// TwinCAT 3 PLC project Horiba
// Title: ZigaLibs.Horiba
// Company: Ziga Javornik
// Author: Ziga Javornik
// ProjectVersion: 0.0.1.0
// Description: Horiba EtherCAT device imeplementations library.
// ProgramVersion: 3.1.4024.0
// libraries:
//   Tc2_Standard, * (Beckhoff Automation GmbH)
//   Tc2_System, * (Beckhoff Automation GmbH)
//   Tc3_Module, * (Beckhoff Automation GmbH)
//   TcUnit, * (www.tcunit.org)
//   ZigaLibs.Automation, * (Ziga)
//   ZigaLibs.Core, * (Ziga)
//   ZigaLibs.Logging, * (Ziga)
// project tree:
//   SOURCE/MFC/SEC_ZXX7/DUTs/ E_SEC_ZXX7_ActuatorControl.TcDUT, E_SEC_ZXX7_ReadingStep.TcDUT, ST_SEC_ZXX7_ActiveExceptions.TcDUT, ST_SEC_ZXX7_CoeList.TcDUT, ST_SEC_ZXX7_Commands.TcDUT, ST_SEC_ZXX7_Feedback.TcDUT, ST_SEC_ZXX7_Inputs.TcDUT, ST_SEC_ZXX7_Outputs.TcDUT, T_SEC_ZXX7_ActiveExceptionStatus.TcDUT, T_SEC_ZXXX7_RampTime.TcDUT
//   SOURCE/MFC/SEC_ZXX7/POUs/ FB_MFC_SEC_ZXX7.TcPOU
//   TESTS/ PRG_TESTS.TcPOU
//   TESTS/Test suites/ FB_SUT_Tests.TcPOU (not stored)
// (motion and I/O tree: see PLC project logging)
// real-time tasks:
//   TASK TestsTask: cycle T#10ms, priority 20, ADS port 350
//   TASK PlcTask: cycle T#10ms, priority 21, ADS port 351

// ---- SOURCE/MFC/SEC_ZXX7/DUTs/E_SEC_ZXX7_ActuatorControl.TcDUT
{attribute 'qualified_only'}
{attribute 'strict'}
TYPE E_SEC_ZXX7_ActuatorControl :
(
	FEEDBACK := 0,
	POSITION := 1,
	FULLY_OPEN := 2,
	FULLY_CLOSE := 3,
	FREEZE_POSITION :=4
)USINT;
END_TYPE

// ---- SOURCE/MFC/SEC_ZXX7/DUTs/E_SEC_ZXX7_ReadingStep.TcDUT
{attribute 'qualified_only'}
{attribute 'strict'}
TYPE E_SEC_ZXX7_ReadingStep :
(
	IDLE,
	GAS_TYPE,
	RATED_FLOW
);
END_TYPE

// ---- SOURCE/MFC/SEC_ZXX7/DUTs/ST_SEC_ZXX7_ActiveExceptions.TcDUT
TYPE ST_SEC_ZXX7_ActiveExceptions :
STRUCT
	DeviceWarning		: BOOL;
	DeviceError			: BOOL;
	ManufacturerWarning	: BOOL;
	ManufacturerError	: BOOL;
END_STRUCT
END_TYPE

// ---- SOURCE/MFC/SEC_ZXX7/DUTs/ST_SEC_ZXX7_CoeList.TcDUT
TYPE ST_SEC_ZXX7_CoeList :
STRUCT
	FluidName	: ZigaLibs_Core.ST_CoeEntry_String128 := (Index := 16#900A, Subindex := 16#04);
	Capacity	: ZigaLibs_Core.ST_CoeEntry_REAL := (Index := 16#900A, SubIndex := 16#06);
END_STRUCT
END_TYPE

// ---- SOURCE/MFC/SEC_ZXX7/DUTs/ST_SEC_ZXX7_Commands.TcDUT
TYPE ST_SEC_ZXX7_Commands EXTENDS ST_MfcCommands :
STRUCT
	RampTime	: T_SEC_ZXXX7_RampTime; // Ramp time setpoint in ms	
	Mode		: E_SEC_ZXX7_ActuatorControl;
END_STRUCT
END_TYPE

// ---- SOURCE/MFC/SEC_ZXX7/DUTs/ST_SEC_ZXX7_Feedback.TcDUT
TYPE ST_SEC_ZXX7_Feedback EXTENDS ST_MfcFeedback :
STRUCT
	ActiveExceptions	: ST_SEC_ZXX7_ActiveExceptions;
END_STRUCT
END_TYPE

// ---- SOURCE/MFC/SEC_ZXX7/DUTs/ST_SEC_ZXX7_Inputs.TcDUT
TYPE ST_SEC_ZXX7_Inputs :
STRUCT
	ValvePosition	: REAL;
	ActualFlow		: REAL;
	ExceptionStatus	: T_SEC_ZXX7_ActiveExceptionStatus;
	AmsAddr			: Tc2_System.ST_AmsAddr;
END_STRUCT
END_TYPE

// ---- SOURCE/MFC/SEC_ZXX7/DUTs/ST_SEC_ZXX7_Outputs.TcDUT
TYPE ST_SEC_ZXX7_Outputs :
STRUCT
	FlowSetpoint	: REAL;
	RampTime		: T_SEC_ZXXX7_RampTime;
	ActuatorControl	: E_SEC_ZXX7_ActuatorControl;
END_STRUCT
END_TYPE

// ---- SOURCE/MFC/SEC_ZXX7/DUTs/T_SEC_ZXX7_ActiveExceptionStatus.TcDUT
TYPE T_SEC_ZXX7_ActiveExceptionStatus : USINT; END_TYPE

// ---- SOURCE/MFC/SEC_ZXX7/DUTs/T_SEC_ZXXX7_RampTime.TcDUT
TYPE T_SEC_ZXXX7_RampTime : UDINT; END_TYPE

// ---- SOURCE/MFC/SEC_ZXX7/POUs/FB_MFC_SEC_ZXX7.TcPOU
FUNCTION_BLOCK FB_MFC_SEC_ZXX7 EXTENDS ZigaLibs_Core.FB_HasInstanceNameAndPath
VAR_INPUT
	commands	: ST_SEC_ZXX7_Commands;	// Commands
	updateCoe	: BOOL;	// Reads COE parameters on rising edge
END_VAR

VAR_OUTPUT
	feedback	: ST_SEC_ZXX7_Feedback;	// Feedback
END_VAR

VAR
	_logger			: REFERENCE TO ZigaLibs_Logging.I_Logger;
	_coeList		: ST_SEC_ZXX7_CoeList;
	_exceptionsPrev	: ST_SEC_ZXX7_ActiveExceptions;
	_sb				: ZigaLibs_Core.FB_StringBuilder;
	_init			: BOOL;
	_readRequest	: Tc2_Standard.R_TRIG;
	_ethercatBoxName		: Tc2_System.T_MaxString;
END_VAR

// IO
VAR
	Inputs	AT %I*	: ST_SEC_ZXX7_Inputs;
	Outputs	AT %Q* 	: ST_SEC_ZXX7_Outputs;
END_VAR

IF NOT commands.Enable THEN
	Outputs.ActuatorControl := E_SEC_ZXX7_ActuatorControl.FULLY_CLOSE;
	Outputs.FlowSetpoint := 0;
ELSE
	Outputs.ActuatorControl := commands.Mode;
	Outputs.FlowSetpoint := commands.FlowSetpoint;
	Outputs.RampTime := commands.RampTime;
END_IF

_readRequest(CLK := updateCoe);
IF _readRequest.Q THEN
	_init := FALSE;
END_IF

IF NOT _init THEN
	THIS^.ReadCoe();
END_IF

feedback.ActiveExceptions.DeviceWarning := Inputs.ExceptionStatus.0;
feedback.ActiveExceptions.DeviceError := Inputs.ExceptionStatus.1;
feedback.ActiveExceptions.ManufacturerWarning := Inputs.ExceptionStatus.2;
feedback.ActiveExceptions.ManufacturerError := Inputs.ExceptionStatus.3;
feedback.ValvePosition := Inputs.ValvePosition;
feedback.ActualFlow := inputs.ActualFlow;

// Error logging
IF __ISVALIDREF(_logger) THEN
	IF feedback.ActiveExceptions.DeviceWarning <> _exceptionsPrev.DeviceWarning THEN
		IF feedback.ActiveExceptions.DeviceWarning THEN
			_logger.LogError(_sb.Reset()
				.AddString(THIS^.GetLogPrefix())
				.AddString('Device warning active!')
				.Create());
		ELSE
			_logger.LogInfo(_sb.Reset()
				.AddString(THIS^.GetLogPrefix())
				.AddString('Device warning no longer active!')
				.Create());			
		END_IF
	END_IF
	
	IF feedback.ActiveExceptions.DeviceError <> _exceptionsPrev.DeviceError THEN
		IF feedback.ActiveExceptions.DeviceError THEN
			_logger.LogError(_sb.Reset()
				.AddString(THIS^.GetLogPrefix())
				.AddString('Device error active!')
				.Create());
		ELSE
			_logger.LogInfo(_sb.Reset()
				.AddString(THIS^.GetLogPrefix())
				.AddString('Device error no longer active!')
				.Create());			
		END_IF
	END_IF
	
	IF feedback.ActiveExceptions.ManufacturerWarning <> _exceptionsPrev.ManufacturerWarning THEN
		IF feedback.ActiveExceptions.ManufacturerWarning THEN
			_logger.LogError(_sb.Reset()
				.AddString(THIS^.GetLogPrefix())
				.AddString('Manufacturer warning active!')
				.Create());
		ELSE
			_logger.LogInfo(_sb.Reset()
				.AddString(THIS^.GetLogPrefix())
				.AddString('Manufacturer warning no longer active!')
				.Create());			
		END_IF
	END_IF
	
	IF feedback.ActiveExceptions.ManufacturerError <> _exceptionsPrev.ManufacturerError THEN
		IF feedback.ActiveExceptions.ManufacturerError THEN
			_logger.LogError(_sb.Reset()
				.AddString(THIS^.GetLogPrefix())
				.AddString('Manufacturer error active!')
				.Create());
		ELSE
			_logger.LogInfo(_sb.Reset()
				.AddString(THIS^.GetLogPrefix())
				.AddString('Manufacturer error no longer active!')
				.Create());			
		END_IF
	END_IF
	
END_IF

_exceptionsPrev := feedback.ActiveExceptions;

{attribute 'hide'}
METHOD FB_init : BOOL
VAR_INPUT
	bInitRetains : BOOL; // if TRUE, the retain variables are initialized (warm start / cold start)
	bInCopyCode : BOOL;  // if TRUE, the instance afterwards gets moved into the copy code (online change)
	logger		: REFERENCE TO ZigaLibs_Logging.I_Logger;
END_VAR
_logger REF= logger;
END_METHOD

{attribute 'monitoring' := 'call'}
// Gets the gas type of the MFC
PROPERTY PUBLIC GasType : STRING(128)
GET
GasType := _coeList.FluidName.Value;
END_GET
END_PROPERTY

METHOD PRIVATE GetLogPrefix : T_MaxString
VAR_INPUT
END_VAR
GetLogPrefix := Tc2_Standard.CONCAT(THIS^.InstancePath, ' - ');
END_METHOD

{attribute 'monitoring' := 'call'}
// Gets the rated flow of the MFC
PROPERTY RatedFlow : REAL
GET
RatedFlow := _coeList.Capacity.Value;
END_GET
END_PROPERTY

METHOD PRIVATE ReadCoe
VAR_INPUT
END_VAR
VAR_INST
	fbCoeReadWrite	: ZigaLibs_Core.FB_CoeReadWrite;
	eCoeReadStep	: E_SEC_ZXX7_ReadingStep;
	bError			: BOOL;
END_VAR
CASE eCoeReadStep OF
	E_SEC_ZXX7_ReadingStep.IDLE:
	IF NOT _init THEN
		IF _ethercatBoxName = '' THEN
				_ethercatBoxName := ZigaLibs_Core.EthercatHelper.GetBoxNameByAddress(
					outError := bError,
					PlcRuntimeNetId := '',
					AmsNetId := Inputs.AmsAddr);
			ELSIF _ethercatBoxName <> '' OR bError THEN
				eCoeReadStep := E_SEC_ZXX7_ReadingStep.GAS_TYPE;
				IF __ISVALIDREF(_logger) THEN
					IF NOT bError THEN
						_logger.LogInfo(message := _sb.Reset()	
							.AddString(str := THIS^.GetLogPrefix())
							.AddString(str := 'Reading CoE parameters for Horiba device ')
							.AddWithDblQuotationMarks(str := _ethercatBoxName)
							.AddString(str := '...')
							.Create());
					ELSE
						_logger.LogInfo(message := _sb.Reset()	
							.AddString(str := THIS^.GetLogPrefix())
							.AddString(str := 'Reading CoE parameters for Horiba device ')
							.AddWithDblQuotationMarks(str := '<Error reading EC box name>')
							.AddString(str := '...')
							.Create());
					END_IF
	
				END_IF
			END_IF
		END_IF
		
	E_SEC_ZXX7_ReadingStep.GAS_TYPE:
		IF fbCoeReadWrite.ReadAny(
				CoeEntry := ADR(_CoeList.FluidName),
				Value := _CoeList.FluidName.Value,
				SlaveAddr := Inputs.AmsAddr)
		THEN
			IF __ISVALIDREF(_logger) THEN
				_logger.LogInfo(_sb.Reset()
					.AddString(THIS^.GetLogPrefix())
					.AddString(' - MFC fluid type is ')
					.AddWithDblQuotationMarks(_coeList.FluidName.Value)
					.Create());
			END_IF
			
			eCoeReadStep := E_SEC_ZXX7_ReadingStep.RATED_FLOW;
		END_IF
		
	E_SEC_ZXX7_ReadingStep.RATED_FLOW:
		IF fbCoeReadWrite.ReadAny(
				CoeEntry := ADR(_CoeList.Capacity),
				Value := _CoeList.Capacity.Value,
				SlaveAddr := Inputs.AmsAddr)
		THEN
			IF __ISVALIDREF(_logger) THEN
				_logger.LogInfo(_sb.Reset()
					.AddString(THIS^.GetLogPrefix())
					.AddString(' - MFC rated flow is ')
					.AddAnyReal(_coeList.Capacity.Value, 3, TRUE)
					.AddString(' sccm.')
					.Create());
			END_IF
			
			eCoeReadStep := E_SEC_ZXX7_ReadingStep.IDLE;
			_init := TRUE;
		END_IF
END_CASE
END_METHOD

END_FUNCTION_BLOCK

// ---- TESTS/PRG_TESTS.TcPOU
PROGRAM PRG_TESTS

(* Instantiate test suites here. Naming convention for tests should be a suffix with _Tests.
Good practice for creating test methods is to end them with _test as well. *)
VAR
	fbSUT_Tests	: FB_SUT_Tests;
END_VAR

// Run tests in parallel
//TcUnit.RUN();

// Run tests in sequence, one after the other.
TcUnit.RUN_IN_SEQUENCE();

END_PROGRAM
